(* Schneider Machine Expert - Basic project Test_Tank, file version 3.0.0.0 *)
(* ProjectInformations: Name=Test_Tank *)

HARDWARE
  Cpu 0: TM221CE24T
  EthernetConfiguration: NetworkName=M221, IpAllocationMode=ByDhcp, IpAddress=192.168.1.10, SubnetMask=255.255.255.0
  SerialLineConfiguration: Baud=Baud19200, Parity=ParityEven, DataBits=DataBits8, StopBits=StopBits1, PhysicalMedium=PhysicalMediumRs485, TransmissionMode=TransmissionModeModbusRtu, SlaveId=1, Addressing=SlaveAddressing
  MastTask: UsePeriodScanMode=false, PeriodScan=100
  FastTask: Period=255
  CpuBehavior: StartingMode=StartAsPreviousState, AutoSaveRamOnEeprom=true, WatchdogPeriod=250

SYMBOLS  (address, symbol, comment, settings)
  %I0.0     LS_TANK1
  %I0.1     LS_TANK2
  %Q0.0     PUMP1
  %Q0.1     PUMP2

POU Test_Tank
  (* SectionNumber=1 *)

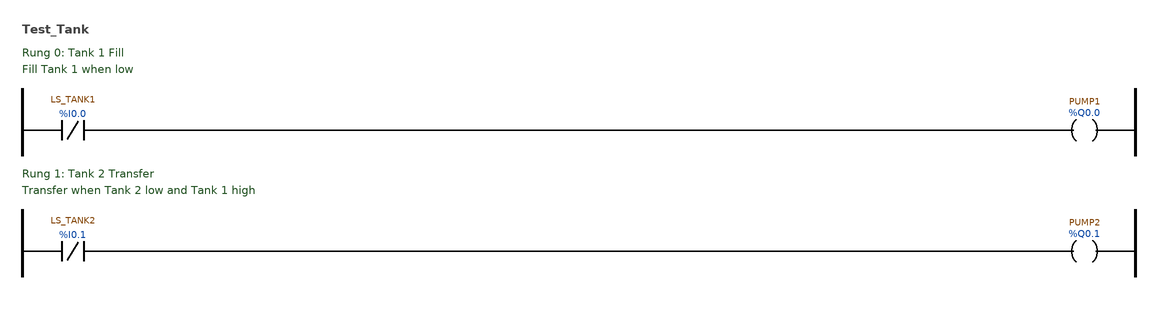

// Rung 0: Tank 1 Fill
// Fill Tank 1 when low
  LDN %I0.0               (* LS_TANK1 *)
  ST %Q0.0                (* PUMP1 *)
  // as ST:
  //   PUMP1 := NOT LS_TANK1;

// Rung 1: Tank 2 Transfer
// Transfer when Tank 2 low and Tank 1 high
  LDN %I0.1               (* LS_TANK2 *)
  ST %Q0.1                (* PUMP2 *)
  // as ST:
  //   PUMP2 := NOT LS_TANK2;
